(* IEC 61131-3 sources: ia2/examples/write_governance/pous, 1 file *)

(* ---- main.st ---- *)
PROGRAM main
VAR
    setpoint : REAL := 0.0;
    observed : REAL := 0.0;
END_VAR
observed := setpoint;
END_PROGRAM
